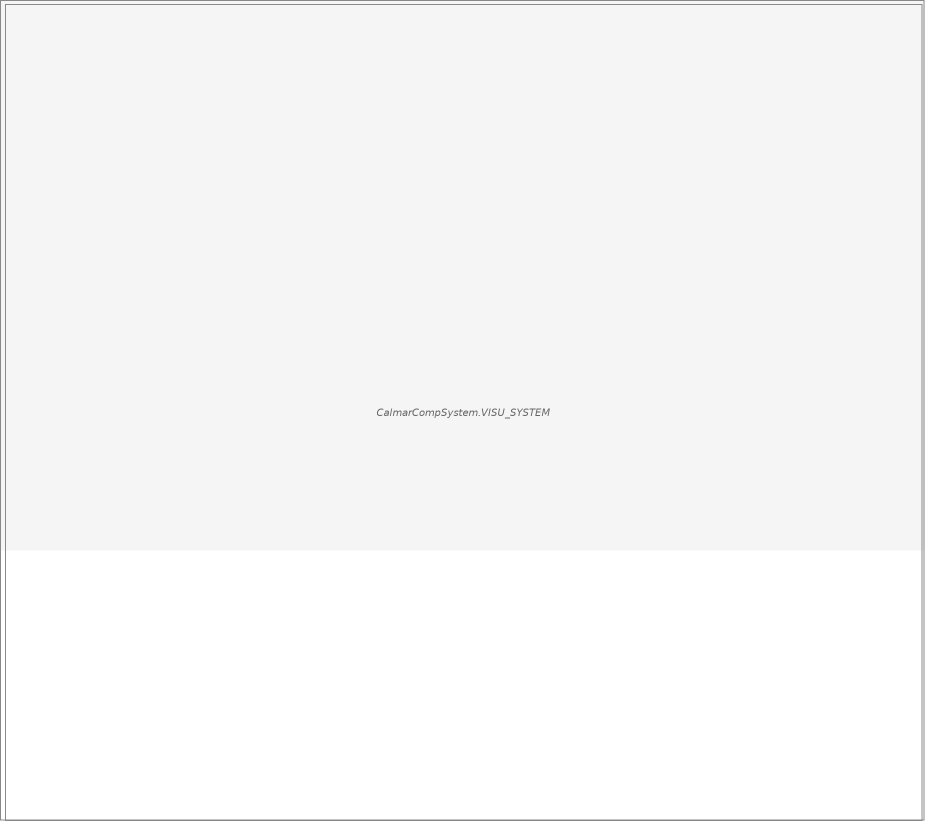
VISUALIZATION VISU_SYSTEM  // 925x821
    Rectangle (0,0 925x550)
    TabControl (5,4 917x817)
        shows CalmarCompSystem.VISU_SYSTEM()
        shows VISU_CANOPEN()
        [1]: TabTitle=CANOpen
END_VISUALIZATION

(* stored: Version 1.1.0.1, ProductVersion 3.1.4024.9
   Visu VISU_SYSTEM: Id {431c0c0c-412b-4cf6-afb5-547ee98aa37e} *)
